INTERFACE IDrilling EXTENDS ZApplication.IUnit

END_INTERFACE

(* stored: Version 1.1.0.1
   Itf IDrilling: Id {0f3e0cad-1965-4457-b473-4fa596cfe2cb} *)
